{attribute 'linkalways'} 
{attribute 'no_explicit_call' := 'This FB is a CLASS and must be accessed using methods or properties'}
{attribute 'enable_dynamic_creation'}
FUNCTION_BLOCK _ETcVnSvmKernelType EXTENDS EnumDatatypeBase
VAR
	localData : ETcVnSvmKernelType;
	activeData : REFERENCE TO ETcVnSvmKernelType;
	enumBaseDatatype : _DINT(localData);
END_VAR

METHOD PRIVATE AddLocalEnumeration
VAR_INPUT
	Enumeration : T_MAXSTRING;
	Value : ETcVnSvmKernelType;
END_VAR
AddEnumeration(Enumeration, Value);
END_METHOD

PROPERTY PUBLIC Address : PVOID
GET
Address := ADR(activeData);
END_GET
END_PROPERTY

METHOD PUBLIC ClearReference
VAR_INPUT
END_VAR
activeData REF= localData;
SetBaseDatatypeReference();
END_METHOD

METHOD PUBLIC Clone : I_Datatype
VAR
    pClone : POINTER TO _ETcVnSvmKernelType;
END_VAR
pClone := __NEW(_ETcVnSvmKernelType(InitialValue := Value));
Clone := pClone^;
END_METHOD

METHOD FB_init : BOOL
VAR_INPUT
	bInitRetains : BOOL; // if TRUE, the retain variables are initialized (warm start / cold start)
	bInCopyCode : BOOL;  // if TRUE, the instance afterwards gets moved into the copy code (online change)
	InitialValue : ETcVnSvmKernelType;
END_VAR
localData := InitialValue;
AddBaseDatatype(enumBaseDatatype);
ClearReference();

AddLocalEnumeration('TCVN_SKT_LINEAR', ETcVnSvmKernelType.TCVN_SKT_LINEAR);
AddLocalEnumeration('TCVN_SKT_POLY', ETcVnSvmKernelType.TCVN_SKT_POLY);
AddLocalEnumeration('TCVN_SKT_RBF', ETcVnSvmKernelType.TCVN_SKT_RBF);
AddLocalEnumeration('TCVN_SKT_SIGMOID', ETcVnSvmKernelType.TCVN_SKT_SIGMOID);
AddLocalEnumeration('TCVN_SKT_CHI2', ETcVnSvmKernelType.TCVN_SKT_CHI2);
AddLocalEnumeration('TCVN_SKT_INTER', ETcVnSvmKernelType.TCVN_SKT_INTER);
END_METHOD

PROPERTY PUBLIC Identifier : T_MAXSTRING
GET
Identifier := 'ETcVnSvmKernelType';
END_GET
END_PROPERTY

METHOD IsEnumeratorValueEqual : BOOL
VAR_INPUT
	Enumerator : I_KeyValueForwardEnumerator;
END_VAR
VAR
	storedValue : ETcVnSvmKernelType;
END_VAR
IF NOT Enumerator.TryGet(storedValue) THEN
	RETURN;
END_IF

IsEnumeratorValueEqual := storedValue = activeData;
END_METHOD

METHOD PUBLIC MakeReferenceTo
VAR_INPUT
	ReferenceTarget : REFERENCE TO ETcVnSvmKernelType;
END_VAR
activeData REF= ReferenceTarget;
SetBaseDatatypeReference();
END_METHOD

METHOD PROTECTED SetBaseDatatypeReference
VAR_INPUT
END_VAR
enumBaseDatatype.MakeReferenceTo(activeData);
END_METHOD

PROPERTY PUBLIC Size : UDINT
GET
Size := SIZEOF(activeData);
END_GET
END_PROPERTY

METHOD TryMakeReferenceTo : BOOL
VAR_INPUT
	Target : I_Datatype;
END_VAR
VAR
	targetAsEnum : I_EnumDatatype;
	pTargetData : POINTER TO ETcVnSvmKernelType;
END_VAR
IF NOT Target.TryResolveAsEnumDatatype(targetAsEnum) THEN
	RETURN;
END_IF

IF targetAsEnum.Identifier <> Identifier THEN
	RETURN;
END_IF

pTargetData := Target.Address;
activeData REF= pTargetData^;
SetBaseDatatypeReference();
TryMakeReferenceTo := TRUE;
END_METHOD

PROPERTY PUBLIC Value : ETcVnSvmKernelType
GET
Value := activeData;
END_GET
SET
activeData := Value;
END_SET
END_PROPERTY

END_FUNCTION_BLOCK

(* stored: Version 1.1.0.1
   POU _ETcVnSvmKernelType: Id {6f92bc58-f9d7-4463-aee5-7a9c2f31b710}, SpecialFunc None
   Folder Constructor: Id {47d69f14-ac61-4ea7-b937-7b540bc73524}
   Folder Private: Id {12ab30b2-833d-4b65-ae8b-a2884510ca01}
   Folder Protected: Id {aff70644-213b-4ea1-8e39-20d4774a9148}
   Method AddLocalEnumeration: Id {0b35c0ea-a634-4493-8f64-076e88c0731d}
   Property Address: Id {025cc496-46ca-463c-bb25-d89a50ae08df}
   Get Get: Id {4bc6dfa9-b505-43a2-9d67-0c14b03aa5e3}
   Method ClearReference: Id {fdfcf6be-fcb5-4b32-a59c-0679ecbb87ce}
   Method Clone: Id {d9c67f80-e0d2-4acd-916d-6406efc0ee62}
   Method FB_init: Id {8d313b60-b134-4ca6-a363-6516183b3022}
   Property Identifier: Id {c71a237e-7b8a-4d62-9542-e604bc8abd72}
   Get Get: Id {36044ff3-a804-435c-92c6-f09bf2c1aa6f}
   Method IsEnumeratorValueEqual: Id {85005c6c-51c6-4e02-bf76-b5aa169c94bb}
   Method MakeReferenceTo: Id {0a8a573d-b67e-4ba5-abc4-31208bc8a513}
   Method SetBaseDatatypeReference: Id {deab7f48-e197-4b52-a08f-4164bad11abf}
   Property Size: Id {d094d822-bcc7-4615-af11-5a0092be4d05}
   Get Get: Id {2ce388f1-5cf5-40b4-aad1-ba609fe95bbf}
   Method TryMakeReferenceTo: Id {ee34c289-ef7c-4d54-ae8c-6595a45b1650}
   Property Value: Id {26301886-4ec7-4bf3-b41b-65dd1adb9dad}
   Get Get: Id {04b18888-105b-4b16-8104-665b81b7be64}
   Set Set: Id {6f4f17ec-05f6-423d-a303-125eae3fbb48} *)
